PROGRAM MAIN
VAR
END_VAR

END_PROGRAM

(* stored: Version 1.1.0.1
   POU MAIN: Id {c6126699-3bb2-471a-b2f7-db9a601914c0} *)
